FUNCTION_BLOCK TankLD
VAR_INPUT
	diMixer_Running : BOOL;
	diMixer_Error : BOOL;
END_VAR
VAR_OUTPUT
	doMixer_Start : BOOL;
END_VAR
VAR_IN_OUT
	ioTank : TTank;
	mixer : Engine;
END_VAR

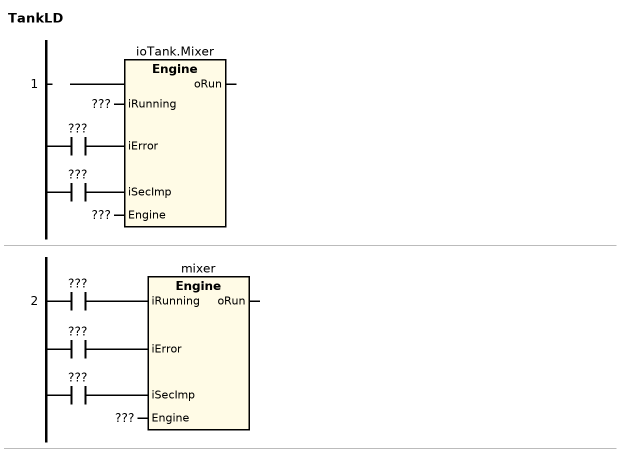
// NETWORK 1
ioTank.Mixer(); // Engine

// NETWORK 2
mixer(); // Engine

END_FUNCTION_BLOCK

(* stored: Version 1.1.0.1, ProductVersion 3.1.4024.12
   POU TankLD: Id {2e1e9142-bdfa-491c-9731-2c8403a98f0e}, SpecialFunc None *)
